(* IEC 61131-3 sources: Industry-PLC-LLM/data/PLCBEAD_repo/PLCBEAD_PLCEmbed-main/PLC-BEAD/Source/GEB/_BYTE_TO_INT, 1 file *)

(* ---- _BYTE_TO_INT.ST ---- *)
FUNCTION _BYTE_TO_INT:INT
	VAR_INPUT
		IN :	BYTE;
	END_VAR

	_BYTE_TO_INT := USINT_TO_INT(BYTE_TO_USINT(IN));
END_FUNCTION

PROGRAM program0
  VAR
    LocalVar0 : BYTE;
	LocalOUT  : INT;
  END_VAR

  LocalOUT := _BYTE_TO_INT(LocalVar0);
END_PROGRAM
